(* IEC 61131-3 sources: plc-vscode/crates/plc_syntax/test_data/parser, 1 file *)

(* ---- malformed_missing_end_program.st ---- *)
PROGRAM Broken
VAR
    Value : BOOL;
END_VAR

FUNCTION_BLOCK StillParsed
END_FUNCTION_BLOCK
